INTERFACE I_StateManager EXTENDS I_Debug, I_Tagged, I_OwnedComp

PROPERTY Current : I_State
GET
END_GET
END_PROPERTY

PROPERTY Pretender : I_State
GET
END_GET
END_PROPERTY

PROPERTY Previous : I_State
GET
END_GET
END_PROPERTY

METHOD Request : Result
VAR_INPUT
	iState		: I_State;
END_VAR
END_METHOD

END_INTERFACE

(* stored: Version 1.1.0.1
   Itf I_StateManager: Id {ec583bc5-9b8d-4fc4-91c2-534454363ae3}
   Folder Request: Id {87840c05-c4d3-4f53-8cbe-0a9fd43b4889}
   Folder State: Id {1e4aeef3-5172-4853-a26a-6057d4b308ba}
   Property Current: Id {9e46e8e5-e078-4315-aaef-86ce15f9d553}
   Get Get: Id {6d438f0f-7238-46a4-a0fd-45c0f7fea2b7}
   Property Pretender: Id {7eee6298-11b0-46df-9f35-ba905e3faca3}
   Get Get: Id {f565b10d-746e-4849-a907-af1498783778}
   Property Previous: Id {c2e1c3ef-1230-46cc-9227-0aa972552cdf}
   Get Get: Id {66a045e0-86b0-4b8b-b205-8eac7ef37dde}
   Method Request: Id {cbf2f16f-b719-4bef-889f-617ff3718c21} *)
